(* Logix 5000 project; controller WWTP_SOLIDS_CLX vendor 1 type 14 code 54 rev 17.2; software revision 17.00; part 6 of 16 *)
(* tags used below, declared in another part *)
   Cfg_ClearPulseT : DINT;   // Time to pulse Out_Clear to clear external totalizer (sec)
   PCmd_ClearTot : BOOL;   // Program Command to Clear Totalizer Qty
   PCmd_StartTot : BOOL;   // Program Command to Start Totalizer
   PCmd_StopTot : BOOL;   // Program Command to Stop Totalizer
   PCmd_ZeroFaultInhibit : BOOL;   // Program Command to Inhibit Zero Fault Alarm
   PCmd_ZeroFaultUninhibit : BOOL;   // Program Command to Uninhibit Zero Fault Alarm
   OCmd_ClearTot : BOOL;   // Operator Command to Clear Totalizer Qty
   OCmd_StartTot : BOOL;   // Operator Command to Start Totalizer
   OCmd_StopTot : BOOL;   // Operator Command to Stop Totalizer
   Rdy_ClearTot : BOOL;   // 1=Ready for OCmd_ClearTot (enables button)
   Rdy_StartTot : BOOL;   // 1=Ready for OCmd_StartTot (enables button)
   Rdy_StopTot : BOOL;   // 1=Ready for OCmd_StopTot (enables button)
   Wrk_ValidONS : BOOL;   // Rate PV goes from Infinite or Not a Number to VALID
(* P_DoseFM, continued *)

ROUTINE Prescan   (* ladder *)
// Clear Ownership, clear "lurking" Commands, all Readies
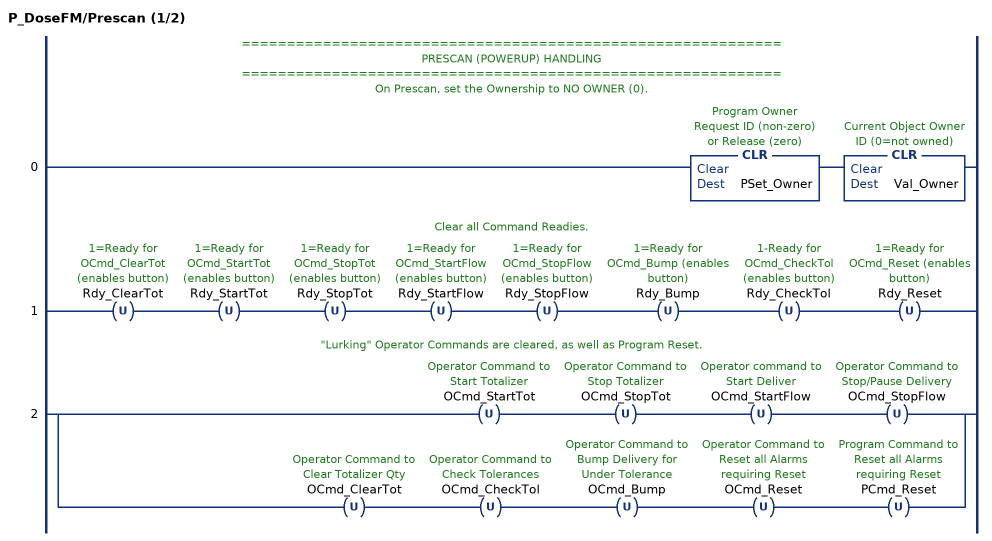
   // ============================================================
   // PRESCAN (POWERUP) HANDLING
   // ============================================================
   // On Prescan, set the Ownership to NO OWNER (0).
   0: CLR(PSet_Owner)CLR(Val_Owner);
   // Clear all Command Readies.
   1: OTU(Rdy_ClearTot)OTU(Rdy_StartTot)OTU(Rdy_StopTot)OTU(Rdy_StartFlow)OTU(Rdy_StopFlow)OTU(Rdy_Bump)OTU(Rdy_CheckTol)OTU(Rdy_Reset);
   // "Lurking" Operator Commands are cleared, as well as Program Reset.
   2: [OTU(OCmd_StartTot) OTU(OCmd_StopTot) OTU(OCmd_StartFlow) OTU(OCmd_StopFlow) ,OTU(OCmd_ClearTot) OTU(OCmd_CheckTol) OTU(OCmd_Bump) OTU(OCmd_Reset) OTU(PCmd_Reset) ];
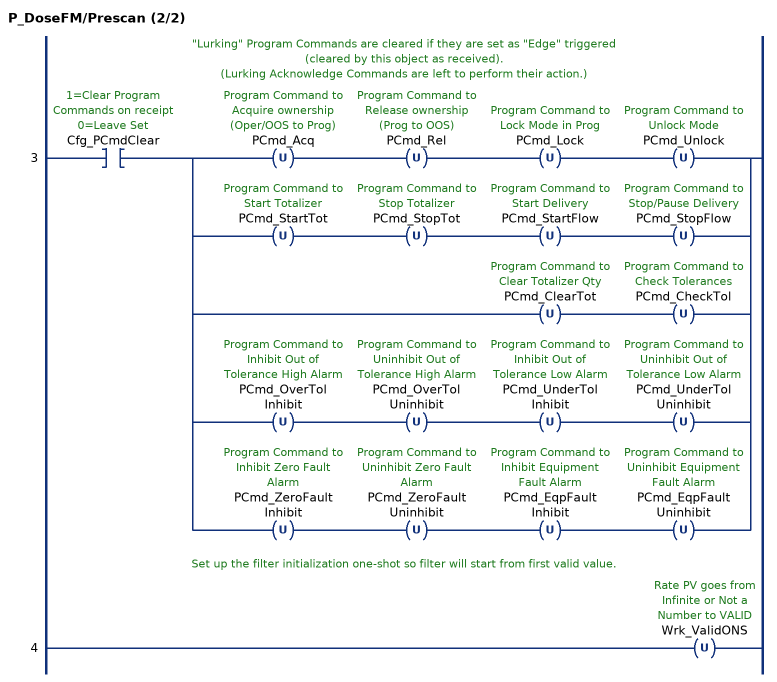
   // "Lurking" Program Commands are cleared if they are set as "Edge" triggered
   // (cleared by this object as received).
   // (Lurking Acknowledge Commands are left to perform their action.)
   3: XIC(Cfg_PCmdClear)[OTU(PCmd_Acq) OTU(PCmd_Rel) OTU(PCmd_Lock) OTU(PCmd_Unlock) ,OTU(PCmd_StartTot) OTU(PCmd_StopTot) OTU(PCmd_StartFlow) OTU(PCmd_StopFlow) ,OTU(PCmd_ClearTot) OTU(PCmd_CheckTol) ,OTU(PCmd_OverTolInhibit) OTU(PCmd_OverTolUninhibit) OTU(PCmd_UnderTolInhibit) OTU(PCmd_UnderTolUninhibit) ,OTU(PCmd_ZeroFaultInhibit) OTU(PCmd_ZeroFaultUninhibit) OTU(PCmd_EqpFaultInhibit) OTU(PCmd_EqpFaultUninhibit) ];
   // Set up the filter initialization one-shot so filter will start from first valid value.
   4: OTU(Wrk_ValidONS);
END_ROUTINE
END_ADD_ON_INSTRUCTION

ADD_ON_INSTRUCTION P_DoseWS   (* revision 0.8, ExecutePrescan, ExecuteEnableInFalse *)
// Dosing with Weigh Scale
// Revision note:
// Fixed handling of Infinite / Not a Number weight PV
// Help:
// This Instruction monitors a weigh scale and provides:
// *  Monitoring of weight rate of change to determine a flow Rate
// *  Command to Tare the scale (set the delivered Quantity to zero)
// *  Commands to Start and Stop Flow for a dosing
// *  Optional switching to a slow delivery (dribble) when approaching setpoint
// *  Stopping flow just before reaching setpoint using a Preact value
// *  Optional automatic adjustment of the preact value to fine tune the stop point
// *  Commands to check if the delivered quantity is within user-specified tolerances and alarm if not
// *  Program and Operator Settings for Setpoint, Preact, Dribble Quantity, High and Low Tolerances
// *  Equipment Failure Alarm on sensor or controlled equipment failure (stops flow)
// *  Tare failure alarm if scale does not stay at steady weight when tared
// *  Configurable Low Rate Cutoff to report zero Rate when scale rate of change is small
// *  Mode selection (Operator, Program or Maintenance)
// *  Simulation using simulated starting weight (Tare point), Running Rate and Dribble Rate
VAR_INPUT
   Inp_WeightPV : REAL; {visible}   // Weight from Weigh Scale (unscaled)
   Inp_PVBad : BOOL;   // 1=Scale PV or I/O Quality Bad, 0=OK
   Inp_PVUncertain : BOOL;   // 1=Scale PV Quality Uncertain, 0=OK
   Inp_CtrldEqpFault : BOOL; {visible}   // Controlled Equipment device or I/O status 0=OK, 1=fail
   Inp_Sim : BOOL;   // 1=Simulate working weigh scale; 0=use actual weight input
   Inp_Reset : BOOL; {visible}   // 1=Reset all fault conditions and latched Alarms
   Cfg_LossInWeight : BOOL;   // 1=Running reduces weight (Xfer Out), 0=iRunning ncreases weight (Xfer In)
   Cfg_HasDribble : BOOL;   // 1=Slow to Dribble before complete, 0=use complete only
   Cfg_AutoAdjPreact : BOOL;   // 1=enable automatic adjustment of preact after each delivery
   Cfg_SetTrack : BOOL := 1;   // 1=PSets track OSets in Oper, OSets track PSets in Prog, 0=no tracking
   Cfg_PCmdClear : BOOL := 1;   // 1=Clear Program Commands on receipt 0=Leave Set
   Cfg_HasOverTolAlm : BOOL;   // 1=Over Tolerance Alarm exists and will be checked
   Cfg_HasUnderTolAlm : BOOL;   // 1=Under Tolerance Alarm exists and will be checked
   Cfg_HasTareFaultAlm : BOOL;   // 1=Tare Fault Alarm exists and will be checked
   Cfg_HasEqpFaultAlm : BOOL;   // 1=Equipment Fault Alarm exists and will be checked
   Cfg_OverTolResetReqd : BOOL;   // 1=Reset requied to clear Out of Tolerance High Alarm
   Cfg_UnderTolResetReqd : BOOL;   // 1=Reset required to clear Out of Tolerance Low Alarm
   Cfg_TareFaultResetReqd : BOOL;   // 1=Reset required to clear Tare Fault Alarm
   Cfg_EqpFaultResetReqd : BOOL;   // 1=Reset required to clear Equipment Fault Alarm
   Cfg_OverTolAckReqd : BOOL := 1;   // 1=Acknowledge required for Out of Tolerance High Alarm
   Cfg_UnderTolAckReqd : BOOL := 1;   // 1=Acknowledge required for Out of Tolerance Low Alarm
   Cfg_TareFaultAckReqd : BOOL := 1;   // 1=Acknowledge required for Tare Fault Alarm
   Cfg_EqpFaultAckReqd : BOOL := 1;   // 1=Acknowledge required for Equipment Fault Alarm
   Cfg_OverTolSeverity : SINT := 3;   // Over Tolerance Alarm Severity 1=info, 2=warn, 3=excep, 4=fault
   Cfg_UnderTolSeverity : SINT := 2;   // Under Tolerance Alarm Severity 1=info, 2=warn, 3=excep, 4=fault
   Cfg_TareFaultSeverity : SINT := 4;   // Tare Fault Alarm Severity 1=info, 2=warn, 3=excep, 4=fault
   Cfg_EqpFaultSeverity : SINT := 4;   // Equipment Fault Alarm Severity 1=info, 2=warn, 3=excep, 4=fault
   Cfg_InpRawMin : REAL;   // Minimum unscaled weight input
   Cfg_InpRawMax : REAL := 10000.0;   // Maximum unscaled weight input
   Cfg_PVEUMin : REAL;   // Minimum scaled weight PV input (EU)
   Cfg_PVEUMax : REAL := 10000.0;   // Maximum scaled weight PV input (EU)
   Cfg_MaxQty : REAL := 1.e+38;   // Maximum allowed quantity to deliver (setpoint) (EU)
   Cfg_RateTime : REAL := 1.0;   // Time factor for rate (60 for /min, 3600 for /hr) (Sec)
   Cfg_RateFiltTC : REAL := 0.1;   // Filter Time Constant (sec) for calculated Rate
   Cfg_TareFaultLim : REAL := 1.0;   // Amount (EU) scale can drift after Tare before starting flow without Faulting
   Cfg_BumpT : REAL := 3.0;   // Bump (manual top-off) Time (Sec)
   Cfg_AutoAdjPct : REAL := 10.0;   // Percentage of delivery error to auto-adjust preact (%)
   Cfg_SimStartWt : REAL;   // Weight to start from (tare to) in simulation (EU)
   Cfg_SimRate : REAL := 1.0;   // Rate at which to deliver when running in Simulation (EU/rate time)
   Cfg_SimDribbleRate : REAL := 0.1;   // Rate at which to dribble when running in Simulation (EU/rate time)
   PSet_SP : REAL;   // Program Setting of total quantity to deliver (EU)
   PSet_DribbleQty : REAL;   // Program Setting of quantity to dribble (EU)
   PSet_Preact : REAL;   // Program Setting of amount before total to stop flow (EU)
   PSet_TolHi : REAL;   // Program Setting of High Tolerance Limit (OK amount > SP)
   PSet_TolLo : REAL;   // Program Setting of Low Tolerance Limit (OK amount < SP)
   PSet_Owner : DINT;   // Program Owner Request ID (non-zero) or Release (zero)
   OSet_SP : REAL;   // Operator Setting of total quantity to deliver (EU)
   OSet_DribbleQty : REAL;   // Operator Setting of quantity to dribble (EU)
   OSet_Preact : REAL;   // Operator Setting of amount before total to stop flow (EU)
   OSet_TolHi : REAL;   // Operator Setting of High Tolerance Limit (OK amount > SP)
   OSet_TolLo : REAL;   // Operator Setting of Low Tolerance Limit (OK amount < SP)
   PCmd_Tare : BOOL;   // Program Command to Tare (reset delivered qty to 0)
   PCmd_StartFlow : BOOL;   // Program Command to Start Delivery
   PCmd_StopFlow : BOOL;   // Program Command to Stop/Pause Delivery
   PCmd_CheckTol : BOOL;   // Program Command to Check Tolerances
   PCmd_Acq : BOOL;   // Program Command to Acquire ownership (Oper/OOS to Prog)
   PCmd_Rel : BOOL;   // Program Command to Release ownership (Prog to OOS)
   PCmd_Lock : BOOL;   // Program Command to Lock Mode in Prog
   PCmd_Unlock : BOOL;   // Program Command to Unlock Mode
   PCmd_Reset : BOOL;   // Program Command to Reset all Alarms requiring Reset
   PCmd_OverTolAck : BOOL;   // Program Command to Acknowledge Out of Tolerance High Alarm
   PCmd_OverTolInhibit : BOOL;   // Program Command to Inhibit Out of Tolerance High Alarm
   PCmd_OverTolUninhibit : BOOL;   // Program Command to Uninhibit Out of Tolerance High Alarm
   PCmd_UnderTolAck : BOOL;   // Program Command to Acknowledge Out of Tolerance Low Alarm
   PCmd_UnderTolInhibit : BOOL;   // Program Command to Inhibit Out of Tolerance Low Alarm
   PCmd_UnderTolUninhibit : BOOL;   // Program Command to Uninhibit Out of Tolerance Low Alarm
   PCmd_TareFaultAck : BOOL;   // Program Command to Acknowledge Tare Fault Alarm
   PCmd_TareFaultInhibit : BOOL;   // Program Command to Inhibit Tare Fault Alarm
   PCmd_TareFaultUninhibit : BOOL;   // Program Command to Uninhibit Tare Fault Alarm
   PCmd_EqpFaultAck : BOOL;   // Program Command to Acknowledge Equipment Fault Alarm
   PCmd_EqpFaultInhibit : BOOL;   // Program Command to Inhibit Equipment Fault Alarm
   PCmd_EqpFaultUninhibit : BOOL;   // Program Command to Uninhibit Equipment Fault Alarm
   OCmd_Tare : BOOL;   // Operator Command to Tare (reset delivered qty to 0)
   OCmd_StartFlow : BOOL;   // Operator command to Start Deliver
   OCmd_StopFlow : BOOL;   // Operator Command to Stop/Pause Delivery
   OCmd_CheckTol : BOOL;   // Operator Command to Check Tolerances
   OCmd_Bump : BOOL;   // Operator Command to Bump Delivery for Under Tolerance
   OCmd_Reset : BOOL;   // Operator Command to Reset all Alarms requiring Reset
END_VAR
VAR_OUTPUT
   Out_RunFlow : BOOL; {visible}   // 1=Deliver at Full (fast) Flow
   Out_DribbleFlow : BOOL; {visible}   // 1=Deliver at Dribble (slow) Flow
   Out_StopFlow : BOOL; {visible}   // 1=Stop Delivery Equipment
   Val_PV : REAL; {visible}   // Weight on Scale (EU)
   Val_Tare : REAL; {visible}   // Weight on Scale when Tare Command received (EU)
   Val_Qty : REAL; {visible}   // Quantity actually delivered (totalizer output) (EU)
   Val_Rate : REAL; {visible}   // Current Delivery Rate (EU/time) (see Cfg_RateTime)
   Val_SP : REAL; {visible}   // Amount to be delivered (Setpoint) (EU)
   Val_Remain : REAL; {visible}   // Amount yet to deliver to reach Setpoint (EU)
   Val_PctComplete : REAL; {visible}   // Percent Complete (for Progress Bar on HMI) 0.0 to 100.0%
   Val_DribbleQty : REAL; {visible}   // Amount to be delivered at slow rate (EU)
   Val_Preact : REAL; {visible}   // Amount before SP at which flow will be stopped (EU)
   Val_TolHi : REAL; {visible}   // Allowed Amount > SP (EU)
   Val_TolLo : REAL; {visible}   // Allowed Amount < SP (EU)
   Val_PVEUMin : REAL;   // Minimum of scaled range = MIN (Cfg_PVEUMin, Cfg_PVEUMax)
   Val_PVEUMax : REAL := 10000.0;   // Maximum of scaled range = MAX (Cfg_PVEUMin, Cfg_PVEUMax)
   Val_Owner : DINT;   // Current Object Owner ID (0=not owned)
   Val_Notify : SINT;   // Current Alarm Level and Acknowledgement (enumeration)
   Sts_Tared : BOOL; {visible}   // Scale Tare completed, Qty = 0.0
   Sts_FlowRunning : BOOL; {visible}   // 1=Flow is Running (Out_Run is ON)
   Sts_FlowDribble : BOOL; {visible}   // 1=Flow is slowed to Dribble (Out_Dribble is ON)
   Sts_FlowStopped : BOOL; {visible}   // 1=Flow is Stopped (Out_Stop is ON)
   Sts_Bumping : BOOL;   // 1=Bump flow (timed) is active
   Sts_Complete : BOOL; {visible}   // 1=Total Delivered > (SP - Preact)
   Sts_InTol : BOOL;   // 1=Total Delivered is Within Tolerances
   Sts_Available : BOOL;   // 1=Dosing available for control by automation (Prog)
   Sts_PVBad : BOOL;   // 1=Weight PV and Rate PV Quality Bad (I/O fail), 0=OK
   Sts_PVUncertain : BOOL;   // 1=Weight PV and Rate PV Quality is Uncertian, 0=OK
   Sts_Err : BOOL; {visible}   // 1=Error: Bad Configuration, see detail Err bits for reason
   Err_Raw : BOOL;   // 1=Error: Cfg_InpRawMax or Cfg_InpRawMin invalid
   Err_EU : BOOL;   // 1=Error: Cfg_PVEUMax or Cfg_PVEUMin invalid
   Err_Rate : BOOL;   // 1=Error: Cfg_RateFiltTC or Cfg_RateTime invalid
   Err_Limit : BOOL;   // 1=Error: Cfg_MaxQty invalid
   Err_Sim : BOOL;   // 1=Error: Cfg_SimDribbleRate or Cfg_SimRate invalid
   Err_Timer : BOOL;   // 1=Error: Cfg_BumpT (use 0.0 to 2147483.647)
   Err_Alarm : BOOL;   // 1=Error: Alarm Min Duration or Severity Cfg Invalid
   Sts_Maint : BOOL; {visible}   // 1=Mode is Maintenance (supersedes Prog, Oper)
   Sts_Prog : BOOL; {visible}   // 1=Mode is Program (auto)
   Sts_Oper : BOOL := 1; {visible}   // 1=Mode is Operator (manual)
   Sts_ProgOperLock : BOOL;   // 1=Program or Operator has requested Mode Lock
   Sts_OverTol : BOOL;   // 1=Delivery Out of Tolerance High
   Alm_OverTol : BOOL;   // 1=Delivery Out of Tolerance High Alarm
   Ack_OverTol : BOOL;   // 1=Out of Tolerance High Alarm has been acknowledged
   Sts_OverTolDisabled : BOOL;   // 1=Out of Tolerance High Alarm has been disabled (will not be sent)
   Sts_OverTolInhibited : BOOL;   // 1=Out of Tolerance High Alarm has been inhibited by logic
   Sts_OverTolSuppressed : BOOL;   // 1=Out of Tolerance High Alarm has been suppressed (logged only)
   Sts_UnderTol : BOOL;   // 1=Delivery Out of Tolerance Low
   Alm_UnderTol : BOOL;   // 1=Delivery Out of Tolerance Low Alarm
   Ack_UnderTol : BOOL;   // 1=Out of Tolerance Low Alarm has been acknowledged
   Sts_UnderTolDisabled : BOOL;   // 1=Out of Tolerance Low Alarm has been disabled (will not be sent)
   Sts_UnderTolInhibited : BOOL;   // 1=Out of Tolerance Low Alarm has been inhibited by logic
   Sts_UnderTolSuppressed : BOOL;   // 1=Out of Tolerance Low Alarm has been suppressed (logged only)
   Sts_TareFault : BOOL;   // 1=Scale reading moved unexpectedly since Tare
   Alm_TareFault : BOOL;   // 1=Warning: scale reading moved since Tare
   Ack_TareFault : BOOL;   // 1=Tare Fault Alarm has been acknowledged
   Sts_TareFaultDisabled : BOOL;   // 1=Tare Fault Alarm is Disabled (not saved or sent)
   Sts_TareFaultInhibited : BOOL;   // 1=Tare Fault Alarm has been inhibited by logic
   Sts_TareFaultSuppressed : BOOL;   // 1=Tare Fault Alarm has been suppressed (logged only)
   Sts_EqpFault : BOOL;   // 1=Equipment Fault Detected
   Alm_EqpFault : BOOL;   // 1=Equipment Fault Alarm
   Ack_EqpFault : BOOL;   // 1=Equipment Fault Alarm has been acknowledged
   Sts_EqpFaultDisabled : BOOL;   // 1=Equipment Fault Alarm is Disabled (not saved or sent)
   Sts_EqpFaultInhibited : BOOL;   // 1=Equipment Fault Alarm has been inhibited by logic
   Sts_EqpFaultSuppressed : BOOL;   // 1=Equipment Fault Alarm has been suppressed (logged only)
   Rdy_Tare : BOOL;   // 1=Ready for OCmd_Tare (enables button)
   Rdy_StartFlow : BOOL;   // 1=Ready for OCmd_StartFlow (enables button)
   Rdy_StopFlow : BOOL;   // 1=Ready for OCmd_StopFlow (enables button)
   Rdy_CheckTol : BOOL;   // 1-Ready for OCmd_CheckTol (enables button)
   Rdy_Bump : BOOL;   // 1=Ready for OCmd_Bump (enables button)
   Rdy_Reset : BOOL;   // 1=Ready for OCmd_Reset (enables button)
END_VAR
VAR
   Cfg_RateEU : STRING_8 := 'kg/sec';   // Engineering Units for Rate (flow) for display on HMI
   Cfg_Tag : STRING_20 := 'P_DoseWS';   // Tagname for display on HMI
   Cfg_Label : STRING_20 := 'Weigh Scale Dosing';   // Label for graphic symbol displayed on HMI
   Cfg_QtyEU : STRING_8 := 'kg';   // Engineering Units for Quantity for display on HMI
   Cfg_Desc : STRING_40 := 'Dosing with Weigh Scale';   // Description for display on HMI
   Wrk_Notify : DINT;   // Buffer for building Val_Notify
   Mode : P_Mode := (Cfg_PCmdClear := 1, Cfg_OvrdOverLock := 1, Sts_Oper := 1, Rdy_Rel := 1, Rdy_AcqLock := 1);   // Analog Input Mode Selection
   Wrk_Tare : BOOL;   // Request to Tare Scale received
   TareFault : P_Alarm := (Inp := 1, Cfg_AckReqd := 1, Cfg_Severity := 3, Ack := 1, Rdy_Disable := 1);   // Scale not holding at point at which Tared Alarm
   UnderTol : P_Alarm := (Inp := 1, Cfg_AckReqd := 1, Cfg_Severity := 3, Ack := 1, Rdy_Disable := 1);   // Final Quantity Below Low Tolerance Alarm
   OverTol : P_Alarm := (Inp := 1, Cfg_AckReqd := 1, Cfg_Severity := 3, Ack := 1, Rdy_Disable := 1);   // Final Quantity Above High Tolerance Alarm
   EqpFault : P_Alarm := (Inp := 1, Cfg_AckReqd := 1, Cfg_Severity := 3, Ack := 1, Rdy_Disable := 1);   // Equipment (Sensor, Controlled Equip.) Fault Alarm
   Wrk_RunFlow : BOOL;   // 1=Flow (full)( should be running
   Wrk_BumpFlow : BOOL;   // Operator requested bump flow to make up Under Tolerance
   Wrk_BumpT : TIMER := (PRE := 3000);   // Bump Timer for shot of flow to make up Under Tolerance
   Wrk_ScanTime : REAL;   // Time since previous scan (sec)
   Wrk_PrevPV : REAL;   // Previous scan's Val_PV value
   Wrk_Rate : REAL;   // Instantaneous Rate based on change in Inp_Qty
   Wrk_AmtToAdd : REAL;   // Amount to add to Quantity this scan based on Rate
   Wrk_PctComplete : REAL;   // Percent Complete calculation intermediate
   Wrk_PV : REAL;   // Working value of Scale Weight (actual or simulated)
   Wrk_TareWt : REAL;   // Weight on scale when Tare Command received
   Wrk_FiltRate : REAL;   // Working register for calculating filtered delivery rate
   Wrk_BumpNoAdj : BOOL;   // Do NOT auto-adjust Preact if flow was Bumped since Tare
   Wrk_ScanT : TIMER := (PRE := 2147483647);   // Scan Timer (milliseconds, always runs)
   Wrk_Alpha : REAL;   // Filter multiplier = (1 / (1+TC/dT) )
   Wrk_InpDINT : DINT;   // Inp_WeightPV check for Infinite or Not A Number
   Wrk_InpInfNaN : BOOL;   // Input Weight is Infinite or NaN
   Wrk_ValidONS1 : BOOL;   // Weight PV goes from Infinite or Not a Number to VALID
   Wrk_ValidONS2 : BOOL;   // Rate goes from Infinite or Not a Number to VALID
END_VAR

ROUTINE EnableInFalse   (* ladder *)
// Clear any "lurking" Commands and all Readies, set NO MODE
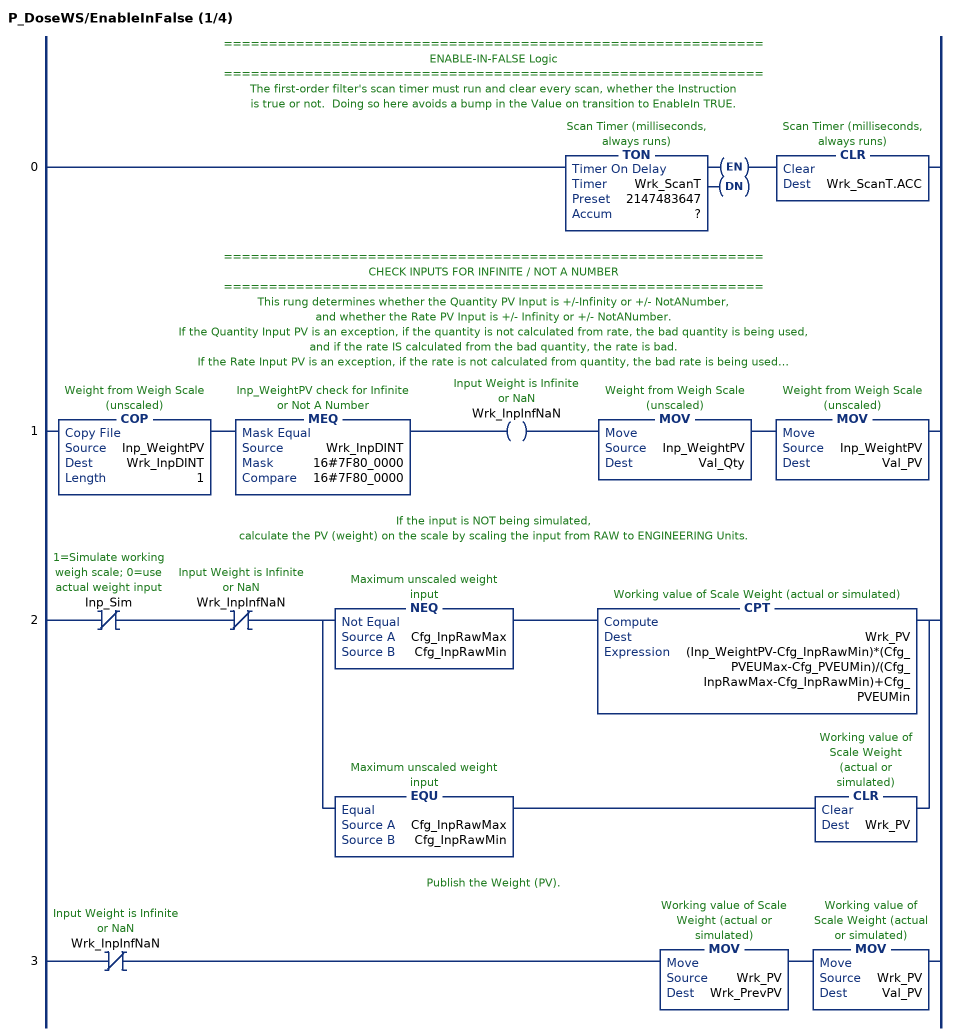
   // ============================================================
   // ENABLE-IN-FALSE Logic
   // ============================================================
   // The first-order filter's scan timer must run and clear every scan, whether the Instruction
   // is true or not.  Doing so here avoids a bump in the Value on transition to EnableIn TRUE.
   0: TON(Wrk_ScanT,?,?)CLR(Wrk_ScanT.ACC);
   // ============================================================
   // CHECK INPUTS FOR INFINITE / NOT A NUMBER
   // ============================================================
   // This rung determines whether the Quantity PV Input is +/-Infinity or +/- NotANumber,
   // and whether the Rate PV Input is +/- Infinity or +/- NotANumber.
   // If the Quantity Input PV is an exception, if the quantity is not calculated from rate, the bad quantity is being used,
   // and if the rate IS calculated from the bad quantity, the rate is bad.
   // If the Rate Input PV is an exception, if the rate is not calculated from quantity, the bad rate is being used,
   // and if the quantity IS calculated from the bad rate, the quantity is bad.
   1: COP(Inp_WeightPV,Wrk_InpDINT,1)MEQ(Wrk_InpDINT,16#7F80_0000,16#7F80_0000)OTE(Wrk_InpInfNaN)MOV(Inp_WeightPV,Val_Qty)MOV(Inp_WeightPV,Val_PV);
   // If the input is NOT being simulated,
   // calculate the PV (weight) on the scale by scaling the input from RAW to ENGINEERING Units.
   2: XIO(Inp_Sim)XIO(Wrk_InpInfNaN)[NEQ(Cfg_InpRawMax,Cfg_InpRawMin) CPT(Wrk_PV,(Inp_WeightPV-Cfg_InpRawMin)*(Cfg_PVEUMax-Cfg_PVEUMin)/(Cfg_InpRawMax-Cfg_InpRawMin)+Cfg_PVEUMin) ,EQU(Cfg_InpRawMax,Cfg_InpRawMin) CLR(Wrk_PV) ];
   // Publish the Weight (PV).
   3: XIO(Wrk_InpInfNaN)MOV(Wrk_PV,Wrk_PrevPV)MOV(Wrk_PV,Val_PV);
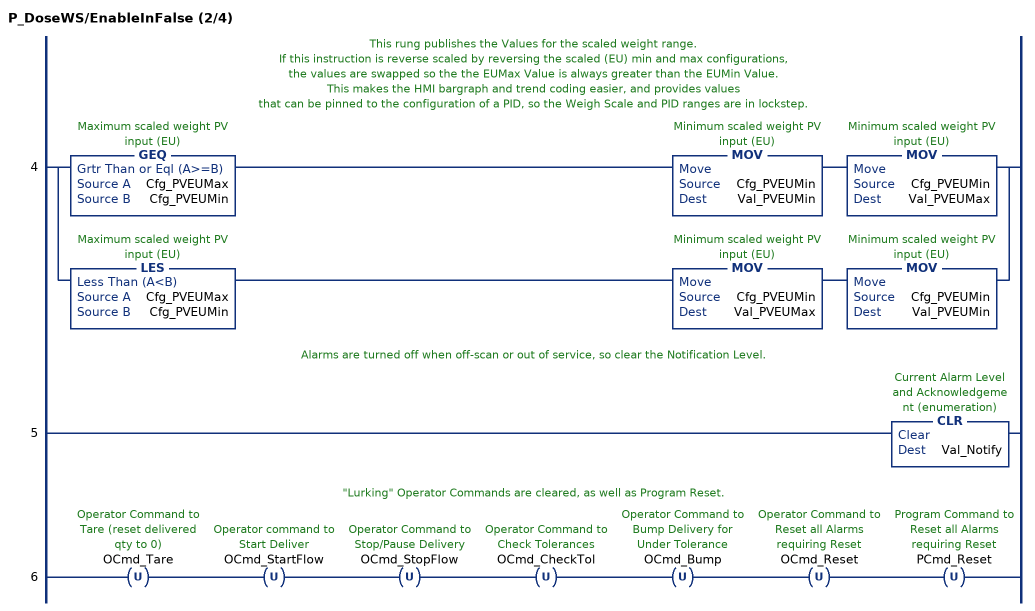
   // This rung publishes the Values for the scaled weight range.
   // If this instruction is reverse scaled by reversing the scaled (EU) min and max configurations,
   // the values are swapped so the the EUMax Value is always greater than the EUMin Value.
   // This makes the HMI bargraph and trend coding easier, and provides values
   // that can be pinned to the configuration of a PID, so the Weigh Scale and PID ranges are in lockstep.
   4: [GEQ(Cfg_PVEUMax,Cfg_PVEUMin) MOV(Cfg_PVEUMin,Val_PVEUMin) MOV(Cfg_PVEUMin,Val_PVEUMax) ,LES(Cfg_PVEUMax,Cfg_PVEUMin) MOV(Cfg_PVEUMin,Val_PVEUMax) MOV(Cfg_PVEUMin,Val_PVEUMin) ];
   // Alarms are turned off when off-scan or out of service, so clear the Notification Level.
   5: CLR(Val_Notify);
   // "Lurking" Operator Commands are cleared, as well as Program Reset.
   6: OTU(OCmd_Tare)OTU(OCmd_StartFlow)OTU(OCmd_StopFlow)OTU(OCmd_CheckTol)OTU(OCmd_Bump)OTU(OCmd_Reset)OTU(PCmd_Reset);
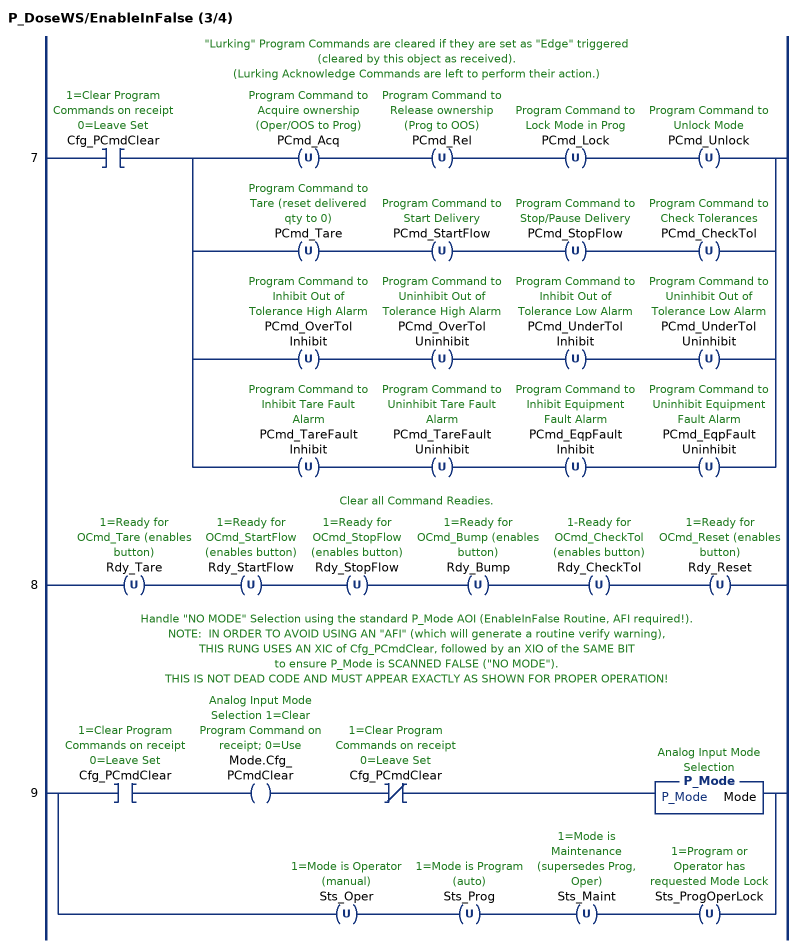
   // "Lurking" Program Commands are cleared if they are set as "Edge" triggered
   // (cleared by this object as received).
   // (Lurking Acknowledge Commands are left to perform their action.)
   7: XIC(Cfg_PCmdClear)[OTU(PCmd_Acq) OTU(PCmd_Rel) OTU(PCmd_Lock) OTU(PCmd_Unlock) ,OTU(PCmd_Tare) OTU(PCmd_StartFlow) OTU(PCmd_StopFlow) OTU(PCmd_CheckTol) ,OTU(PCmd_OverTolInhibit) OTU(PCmd_OverTolUninhibit) OTU(PCmd_UnderTolInhibit) OTU(PCmd_UnderTolUninhibit) ,OTU(PCmd_TareFaultInhibit) OTU(PCmd_TareFaultUninhibit) OTU(PCmd_EqpFaultInhibit) OTU(PCmd_EqpFaultUninhibit) ];
   // Clear all Command Readies.
   8: OTU(Rdy_Tare)OTU(Rdy_StartFlow)OTU(Rdy_StopFlow)OTU(Rdy_Bump)OTU(Rdy_CheckTol)OTU(Rdy_Reset);
   // Handle "NO MODE" Selection using the standard P_Mode AOI (EnableInFalse Routine, AFI required!).
   // NOTE:  IN ORDER TO AVOID USING AN "AFI" (which will generate a routine verify warning),
   // THIS RUNG USES AN XIC of Cfg_PCmdClear, followed by an XIO of the SAME BIT
   // to ensure P_Mode is SCANNED FALSE ("NO MODE").
   // THIS IS NOT DEAD CODE AND MUST APPEAR EXACTLY AS SHOWN FOR PROPER OPERATION!
   9: [XIC(Cfg_PCmdClear) OTE(Mode.Cfg_PCmdClear) XIO(Cfg_PCmdClear) P_Mode(Mode) ,OTU(Sts_Oper) OTU(Sts_Prog) OTU(Sts_Maint) OTU(Sts_ProgOperLock) ];
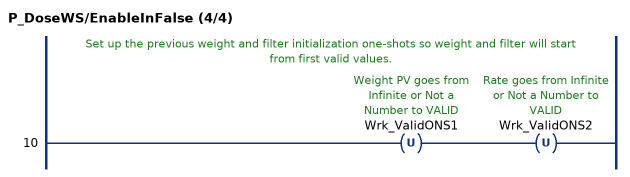
   // Set up the previous weight and filter initialization one-shots so weight and filter will start from first valid values.
   10: OTU(Wrk_ValidONS1)OTU(Wrk_ValidONS2);
END_ROUTINE

ROUTINE Logic   (* ladder *)
// Normal Scan: control / monitor Dosing with Weigh Scale
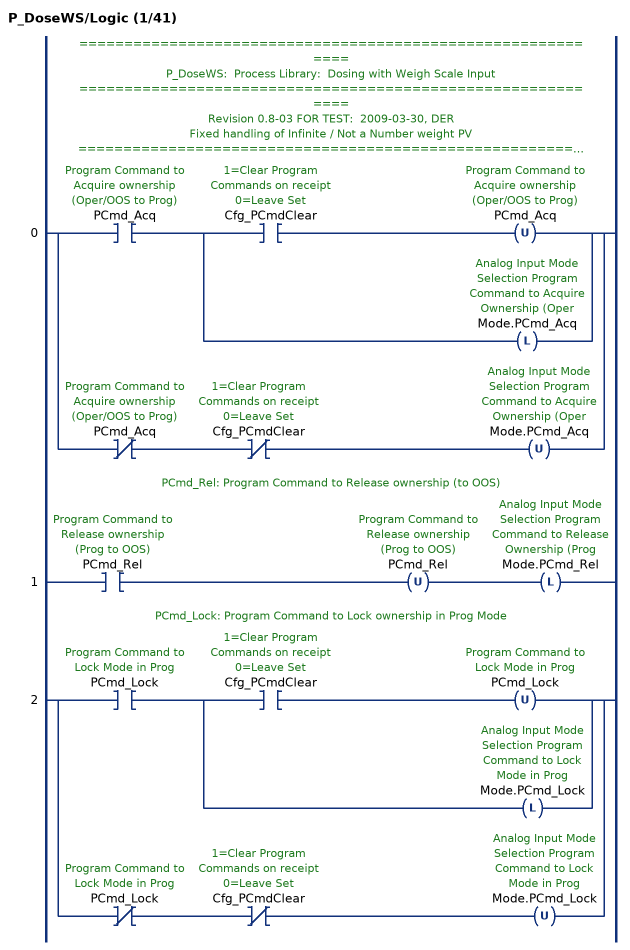
   // ============================================================
   // P_DoseWS:  Process Library:  Dosing with Weigh Scale Input
   // ============================================================
   // Revision 0.8-03 FOR TEST:  2009-03-30, DER
   // Fixed handling of Infinite / Not a Number weight PV
   // ============================================================
   // This Instruction monitors a weigh scale and provides:
   // *  Monitor weight rate of change to determine a flow Rate
   // *  Command to Tare the scale (set the delivered Quantity to zero)
   // *  Commands to Start and Stop Flow for a dosing
   // *  Optional switching to a slow delivery (dribble) when approaching setpoint
   // *  Stopping flow just before reaching setpoint using a Preact value
   // *  Optional automatic adjustment of the preact value to fine tune the stop point
   // *  Commands to check if the delivered quantity is within user-specified tolerances and alarm if not
   // *  Program and Operator Settings for Setpoint, Preact, Dribble Quantity, High and Low Tolerances
   // *  Equipment Failure Alarm on sensor or controlled equipment failure (stops flow)
   // *  Tare failure alarm if scale does not stay at steady weight when tared
   // *  Configurable Low Rate Cutoff to report zero Rate when scale rate of change is small
   // *  Mode selection (Operator, Program or Maintenance)
   // *  Simulation using a provided simulated Tare point, Running Rate and Dribble Rate
   // ============================================================
   // POWERUP / INVALID STATE HANDLING
   // ============================================================
   // See the Prescan routine for powerup handling.
   // Mode states are retained through a power cycle.
   // ============================================================
   // MODE PROCESSING
   // ============================================================
   // These rungs handle received Mode Inputs and Commands:
   // NOTE:  Operator Commands for Mode, Alarm are sent directly to the contained P_Mode and P_Alarm AOIs.
   // PCmd_Acq: Program Command to Acquire ownership
   0: [XIC(PCmd_Acq) [XIC(Cfg_PCmdClear) OTU(PCmd_Acq) ,OTL(Mode.PCmd_Acq) ] ,XIO(PCmd_Acq) XIO(Cfg_PCmdClear) OTU(Mode.PCmd_Acq) ];
   // PCmd_Rel: Program Command to Release ownership (to OOS)
   1: XIC(PCmd_Rel)OTU(PCmd_Rel)OTL(Mode.PCmd_Rel);
   // PCmd_Lock: Program Command to Lock ownership in Prog Mode
   2: [XIC(PCmd_Lock) [XIC(Cfg_PCmdClear) OTU(PCmd_Lock) ,OTL(Mode.PCmd_Lock) ] ,XIO(PCmd_Lock) XIO(Cfg_PCmdClear) OTU(Mode.PCmd_Lock) ];
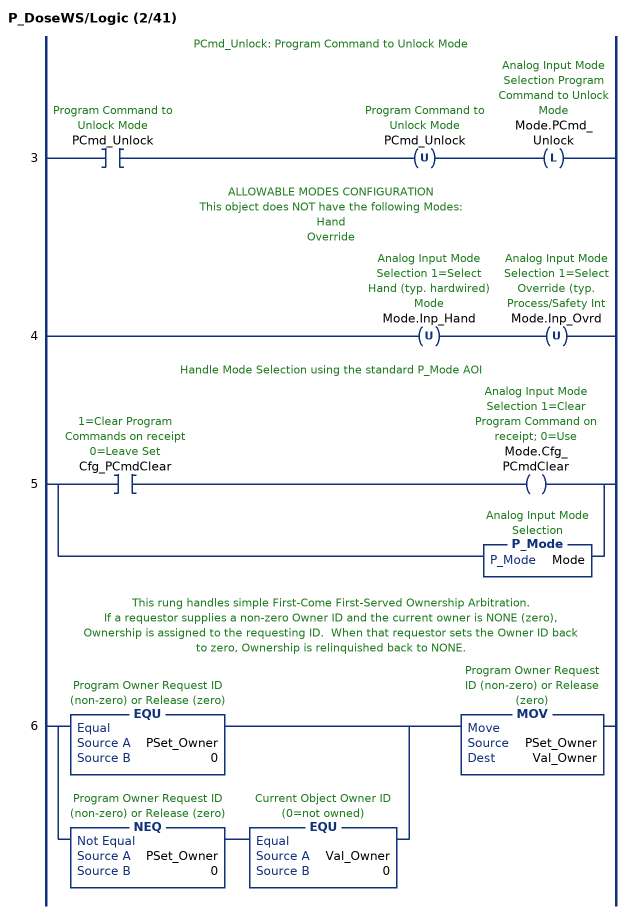
   // PCmd_Unlock: Program Command to Unlock Mode
   3: XIC(PCmd_Unlock)OTU(PCmd_Unlock)OTL(Mode.PCmd_Unlock);
   // ALLOWABLE MODES CONFIGURATION
   // This object does NOT have the following Modes:
   // Hand
   // Override
   4: OTU(Mode.Inp_Hand)OTU(Mode.Inp_Ovrd);
   // Handle Mode Selection using the standard P_Mode AOI
   5: [XIC(Cfg_PCmdClear) OTE(Mode.Cfg_PCmdClear) ,P_Mode(Mode) ];
   // This rung handles simple First-Come First-Served Ownership Arbitration.
   // If a requestor supplies a non-zero Owner ID and the current owner is NONE (zero),
   // Ownership is assigned to the requesting ID.  When that requestor sets the Owner ID back
   // to zero, Ownership is relinquished back to NONE.
   6: [EQU(PSet_Owner,0) ,NEQ(PSet_Owner,0) EQU(Val_Owner,0) ]MOV(PSet_Owner,Val_Owner);
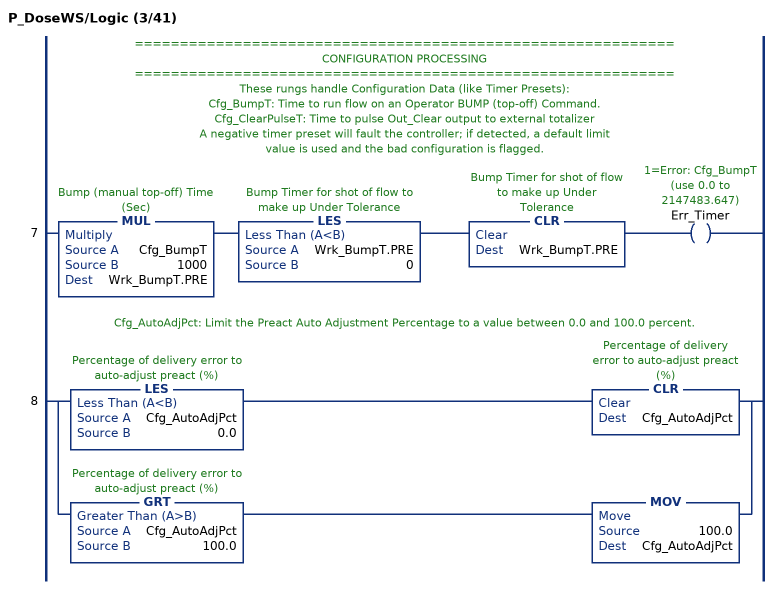
   // ============================================================
   // CONFIGURATION PROCESSING
   // ============================================================
   // These rungs handle Configuration Data (like Timer Presets):
   // Cfg_BumpT: Time to run flow on an Operator BUMP (top-off) Command.
   // Cfg_ClearPulseT: Time to pulse Out_Clear output to external totalizer
   // A negative timer preset will fault the controller; if detected, a default limit
   // value is used and the bad configuration is flagged.
   7: MUL(Cfg_BumpT,1000,Wrk_BumpT.PRE)LES(Wrk_BumpT.PRE,0)CLR(Wrk_BumpT.PRE)OTE(Err_Timer);
   // Cfg_AutoAdjPct: Limit the Preact Auto Adjustment Percentage to a value between 0.0 and 100.0 percent.
   8: [LES(Cfg_AutoAdjPct,0.0) CLR(Cfg_AutoAdjPct) ,GRT(Cfg_AutoAdjPct,100.0) MOV(100.0,Cfg_AutoAdjPct) ];
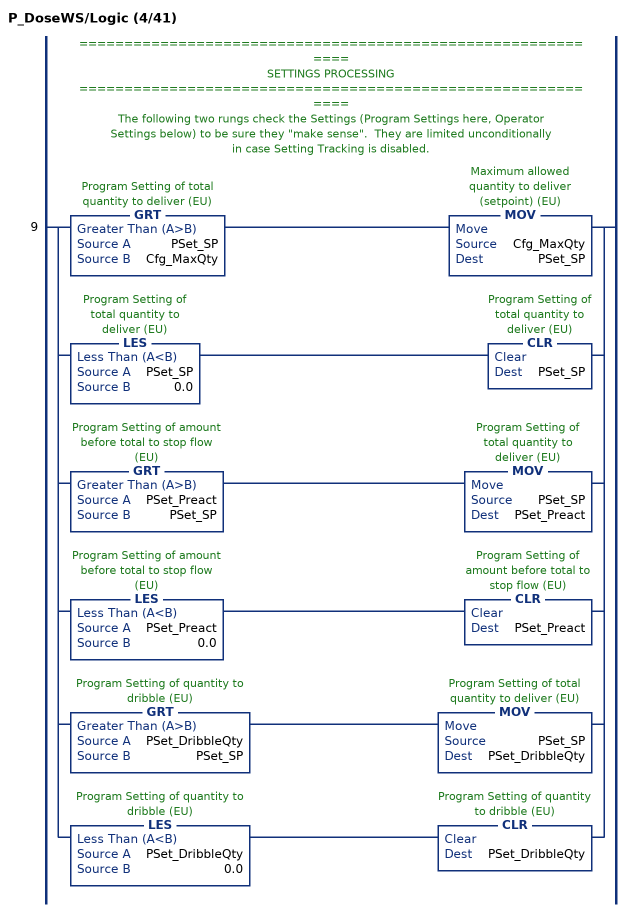
   // ============================================================
   // SETTINGS PROCESSING
   // ============================================================
   // The following two rungs check the Settings (Program Settings here, Operator
   // Settings below) to be sure they "make sense".  They are limited unconditionally
   // in case Setting Tracking is disabled.
   9: [GRT(PSet_SP,Cfg_MaxQty) MOV(Cfg_MaxQty,PSet_SP) ,LES(PSet_SP,0.0) CLR(PSet_SP) ,GRT(PSet_Preact,PSet_SP) MOV(PSet_SP,PSet_Preact) ,LES(PSet_Preact,0.0) CLR(PSet_Preact) ,GRT(PSet_DribbleQty,PSet_SP) MOV(PSet_SP,PSet_DribbleQty) ,LES(PSet_DribbleQty,0.0) CLR(PSet_DribbleQty) ];
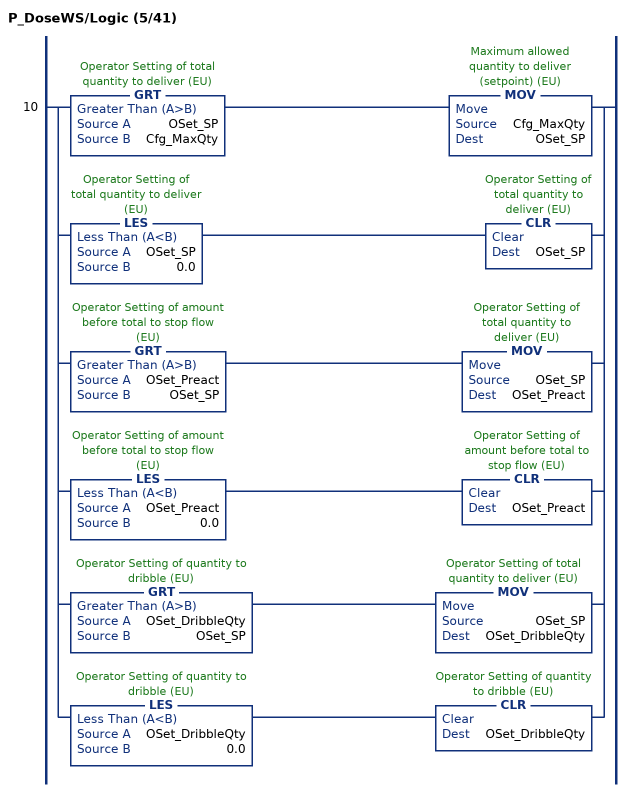
   10: [GRT(OSet_SP,Cfg_MaxQty) MOV(Cfg_MaxQty,OSet_SP) ,LES(OSet_SP,0.0) CLR(OSet_SP) ,GRT(OSet_Preact,OSet_SP) MOV(OSet_SP,OSet_Preact) ,LES(OSet_Preact,0.0) CLR(OSet_Preact) ,GRT(OSet_DribbleQty,OSet_SP) MOV(OSet_SP,OSet_DribbleQty) ,LES(OSet_DribbleQty,0.0) CLR(OSet_DribbleQty) ];
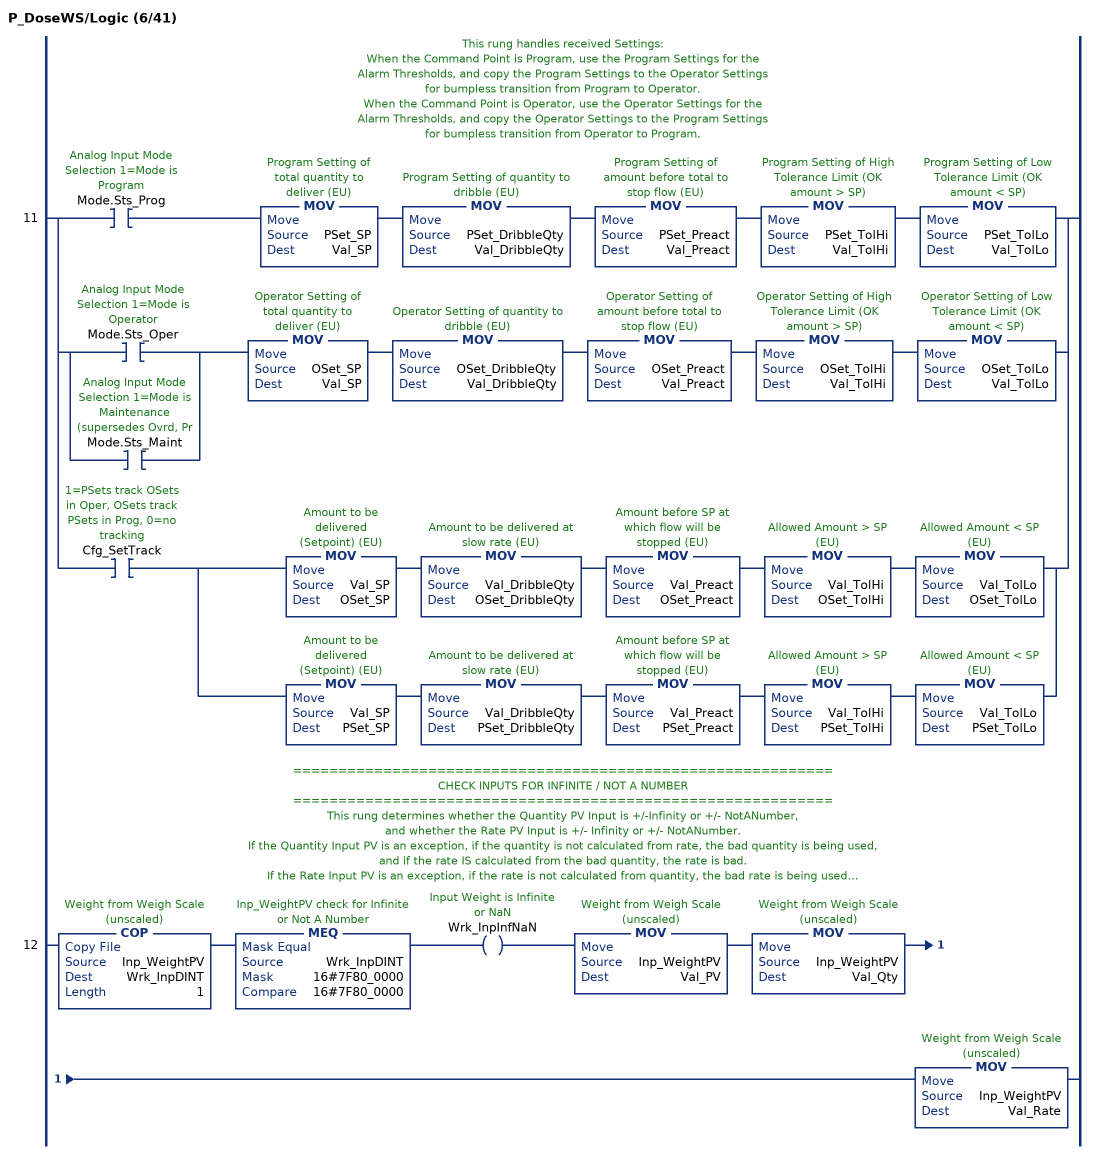
   // This rung handles received Settings:
   // When the Command Point is Program, use the Program Settings for the
   // Alarm Thresholds, and copy the Program Settings to the Operator Settings
   // for bumpless transition from Program to Operator.
   // When the Command Point is Operator, use the Operator Settings for the
   // Alarm Thresholds, and copy the Operator Settings to the Program Settings
   // for bumpless transition from Operator to Program.
   11: [XIC(Mode.Sts_Prog) MOV(PSet_SP,Val_SP) MOV(PSet_DribbleQty,Val_DribbleQty) MOV(PSet_Preact,Val_Preact) MOV(PSet_TolHi,Val_TolHi) MOV(PSet_TolLo,Val_TolLo) ,[XIC(Mode.Sts_Oper) ,XIC(Mode.Sts_Maint) ] MOV(OSet_SP,Val_SP) MOV(OSet_DribbleQty,Val_DribbleQty) MOV(OSet_Preact,Val_Preact) MOV(OSet_TolHi,Val_TolHi) MOV(OSet_TolLo,Val_TolLo) ,XIC(Cfg_SetTrack) [MOV(Val_SP,OSet_SP) MOV(Val_DribbleQty,OSet_DribbleQty) MOV(Val_Preact,OSet_Preact) MOV(Val_TolHi,OSet_TolHi) MOV(Val_TolLo,OSet_TolLo) ,MOV(Val_SP,PSet_SP) MOV(Val_DribbleQty,PSet_DribbleQty) MOV(Val_Preact,PSet_Preact) MOV(Val_TolHi,PSet_TolHi) MOV(Val_TolLo,PSet_TolLo) ] ];
   // ============================================================
   // CHECK INPUTS FOR INFINITE / NOT A NUMBER
   // ============================================================
   // This rung determines whether the Quantity PV Input is +/-Infinity or +/- NotANumber,
   // and whether the Rate PV Input is +/- Infinity or +/- NotANumber.
   // If the Quantity Input PV is an exception, if the quantity is not calculated from rate, the bad quantity is being used,
   // and if the rate IS calculated from the bad quantity, the rate is bad.
   // If the Rate Input PV is an exception, if the rate is not calculated from quantity, the bad rate is being used,
   // and if the quantity IS calculated from the bad rate, the quantity is bad.
   12: COP(Inp_WeightPV,Wrk_InpDINT,1)MEQ(Wrk_InpDINT,16#7F80_0000,16#7F80_0000)OTE(Wrk_InpInfNaN)MOV(Inp_WeightPV,Val_PV)MOV(Inp_WeightPV,Val_Qty)MOV(Inp_WeightPV,Val_Rate);
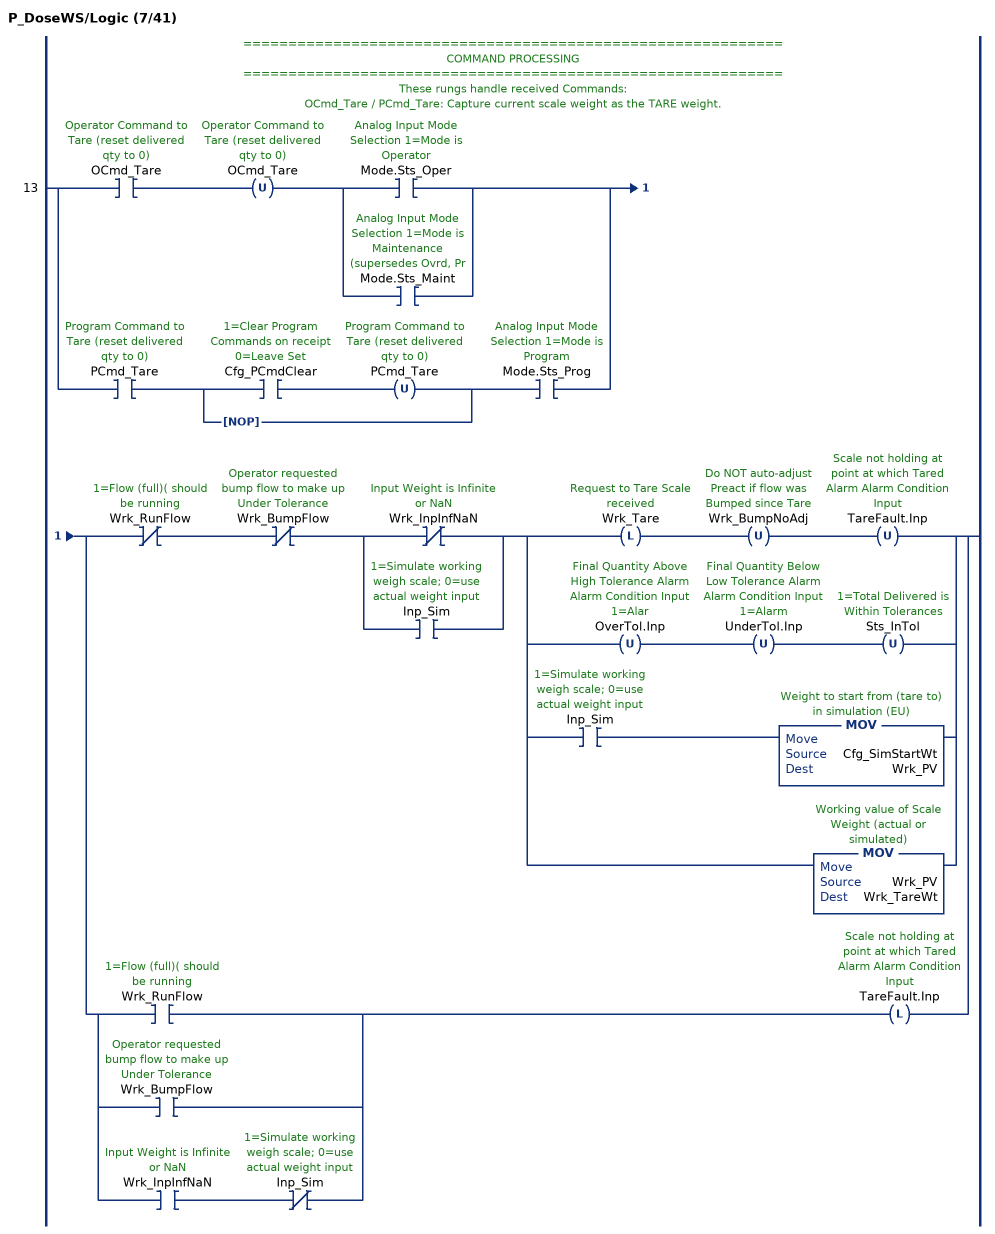
   // ============================================================
   // COMMAND PROCESSING
   // ============================================================
   // These rungs handle received Commands:
   // OCmd_Tare / PCmd_Tare: Capture current scale weight as the TARE weight.
   13: [XIC(OCmd_Tare) OTU(OCmd_Tare) [XIC(Mode.Sts_Oper) ,XIC(Mode.Sts_Maint) ] ,XIC(PCmd_Tare) [XIC(Cfg_PCmdClear) OTU(PCmd_Tare) ,NOP() ] XIC(Mode.Sts_Prog) ][XIO(Wrk_RunFlow) XIO(Wrk_BumpFlow) [XIO(Wrk_InpInfNaN) ,XIC(Inp_Sim) ] [OTL(Wrk_Tare) OTU(Wrk_BumpNoAdj) OTU(TareFault.Inp) ,OTU(OverTol.Inp) OTU(UnderTol.Inp) OTU(Sts_InTol) ,XIC(Inp_Sim) MOV(Cfg_SimStartWt,Wrk_PV) ,MOV(Wrk_PV,Wrk_TareWt) ] ,[XIC(Wrk_RunFlow) ,XIC(Wrk_BumpFlow) ,XIC(Wrk_InpInfNaN) XIO(Inp_Sim) ] OTL(TareFault.Inp) ];
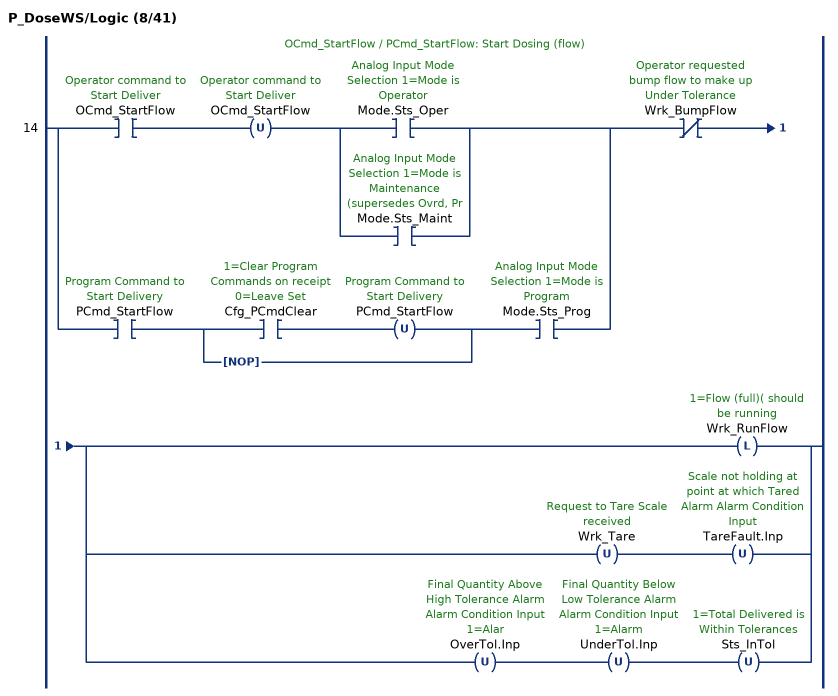
   // OCmd_StartFlow / PCmd_StartFlow: Start Dosing (flow)
   14: [XIC(OCmd_StartFlow) OTU(OCmd_StartFlow) [XIC(Mode.Sts_Oper) ,XIC(Mode.Sts_Maint) ] ,XIC(PCmd_StartFlow) [XIC(Cfg_PCmdClear) OTU(PCmd_StartFlow) ,NOP() ] XIC(Mode.Sts_Prog) ]XIO(Wrk_BumpFlow)[OTL(Wrk_RunFlow) ,OTU(Wrk_Tare) OTU(TareFault.Inp) ,OTU(OverTol.Inp) OTU(UnderTol.Inp) OTU(Sts_InTol) ];
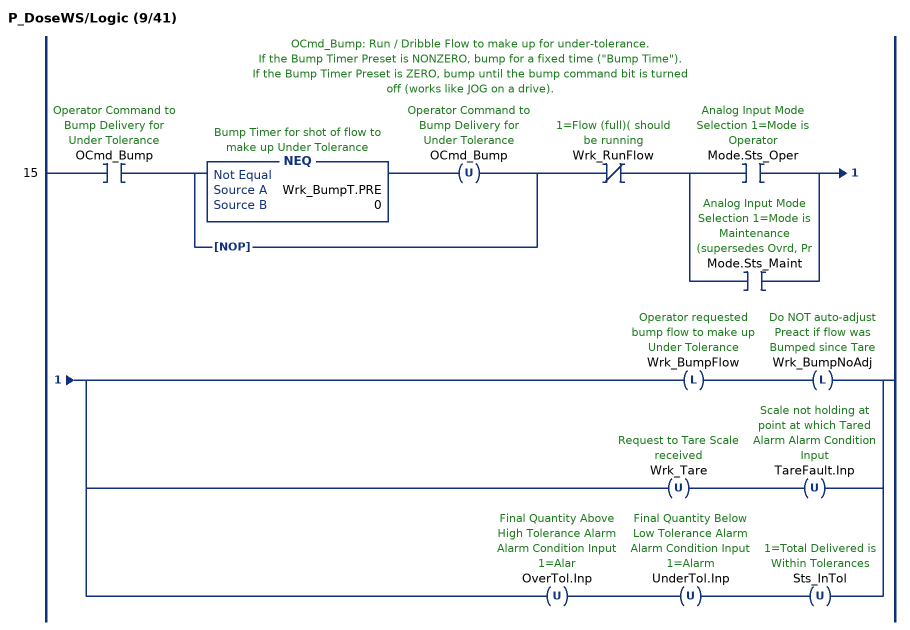
   // OCmd_Bump: Run / Dribble Flow to make up for under-tolerance.
   // If the Bump Timer Preset is NONZERO, bump for a fixed time ("Bump Time").
   // If the Bump Timer Preset is ZERO, bump until the bump command bit is turned
   // off (works like JOG on a drive).
   15: XIC(OCmd_Bump)[NEQ(Wrk_BumpT.PRE,0) OTU(OCmd_Bump) ,NOP() ]XIO(Wrk_RunFlow)[XIC(Mode.Sts_Oper) ,XIC(Mode.Sts_Maint) ][OTL(Wrk_BumpFlow) OTL(Wrk_BumpNoAdj) ,OTU(Wrk_Tare) OTU(TareFault.Inp) ,OTU(OverTol.Inp) OTU(UnderTol.Inp) OTU(Sts_InTol) ];
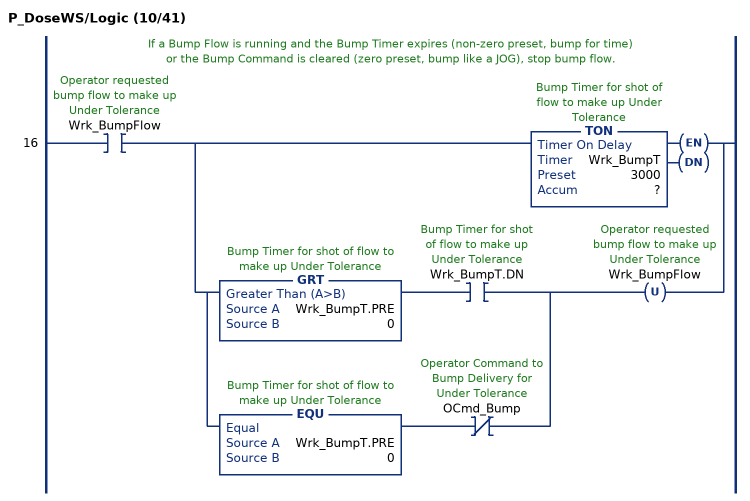
   // If a Bump Flow is running and the Bump Timer expires (non-zero preset, bump for time)
   // or the Bump Command is cleared (zero preset, bump like a JOG), stop bump flow.
   16: XIC(Wrk_BumpFlow)[TON(Wrk_BumpT,?,?) ,[GRT(Wrk_BumpT.PRE,0) XIC(Wrk_BumpT.DN) ,EQU(Wrk_BumpT.PRE,0) XIO(OCmd_Bump) ] OTU(Wrk_BumpFlow) ];
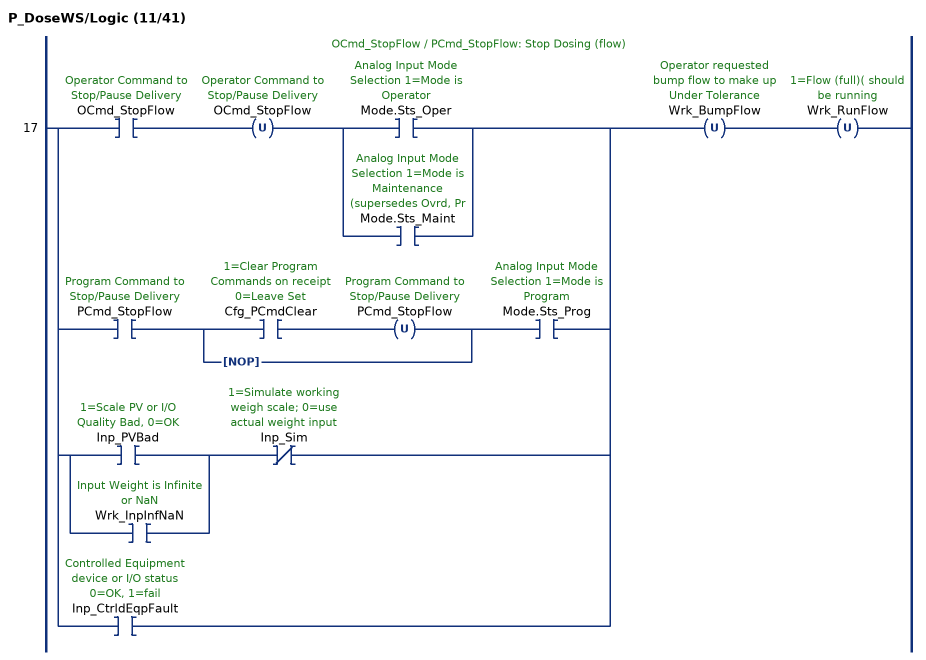
   // OCmd_StopFlow / PCmd_StopFlow: Stop Dosing (flow)
   17: [XIC(OCmd_StopFlow) OTU(OCmd_StopFlow) [XIC(Mode.Sts_Oper) ,XIC(Mode.Sts_Maint) ] ,XIC(PCmd_StopFlow) [XIC(Cfg_PCmdClear) OTU(PCmd_StopFlow) ,NOP() ] XIC(Mode.Sts_Prog) ,[XIC(Inp_PVBad) ,XIC(Wrk_InpInfNaN) ] XIO(Inp_Sim) ,XIC(Inp_CtrldEqpFault) ]OTU(Wrk_BumpFlow)OTU(Wrk_RunFlow);
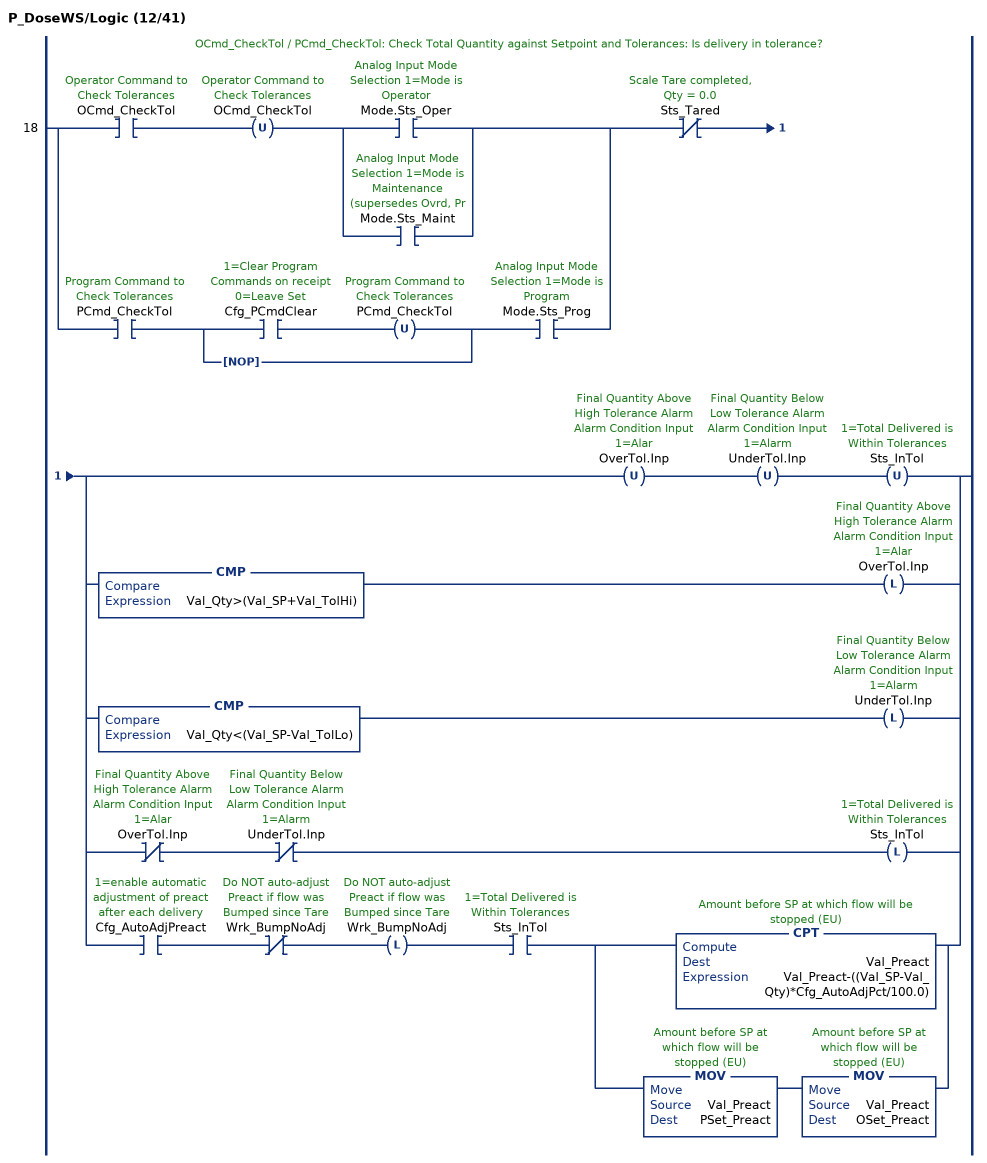
   // OCmd_CheckTol / PCmd_CheckTol: Check Total Quantity against Setpoint and Tolerances: Is delivery in tolerance?
   18: [XIC(OCmd_CheckTol) OTU(OCmd_CheckTol) [XIC(Mode.Sts_Oper) ,XIC(Mode.Sts_Maint) ] ,XIC(PCmd_CheckTol) [XIC(Cfg_PCmdClear) OTU(PCmd_CheckTol) ,NOP() ] XIC(Mode.Sts_Prog) ]XIO(Sts_Tared)[OTU(OverTol.Inp) OTU(UnderTol.Inp) OTU(Sts_InTol) ,CMP(Val_Qty>(Val_SP+Val_TolHi)) OTL(OverTol.Inp) ,CMP(Val_Qty<(Val_SP-Val_TolLo)) OTL(UnderTol.Inp) ,XIO(OverTol.Inp) XIO(UnderTol.Inp) OTL(Sts_InTol) ,XIC(Cfg_AutoAdjPreact) XIO(Wrk_BumpNoAdj) OTL(Wrk_BumpNoAdj) XIC(Sts_InTol) [CPT(Val_Preact,Val_Preact-((Val_SP-Val_Qty)*Cfg_AutoAdjPct/100.0)) ,MOV(Val_Preact,PSet_Preact) MOV(Val_Preact,OSet_Preact) ] ];
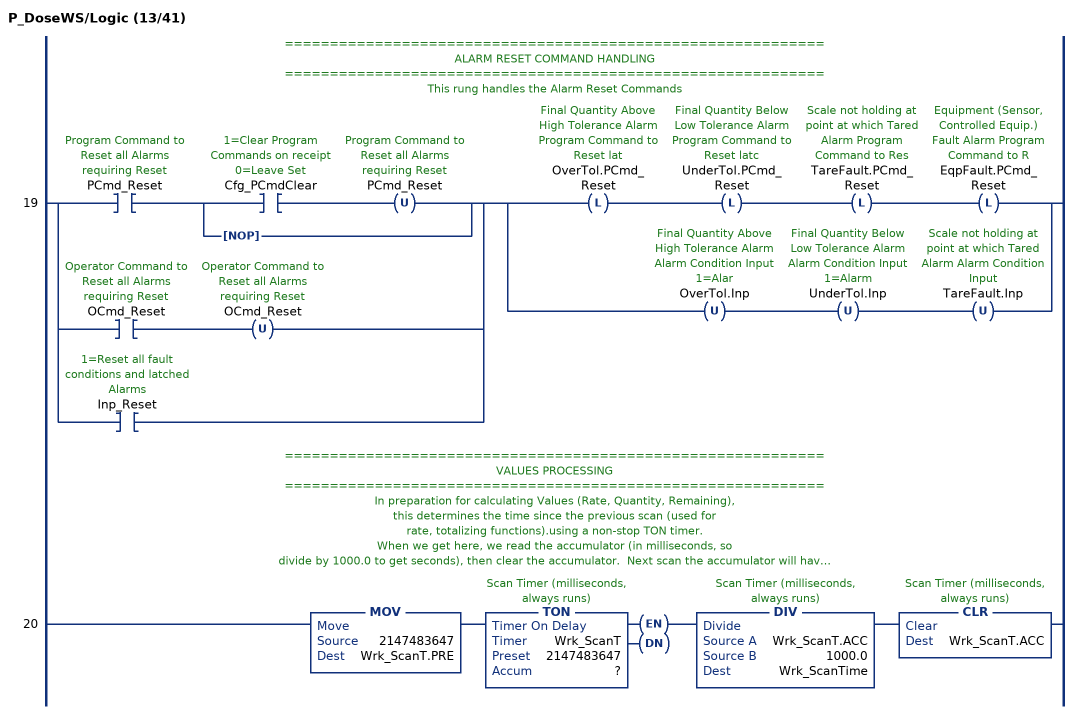
   // ============================================================
   // ALARM RESET COMMAND HANDLING
   // ============================================================
   // This rung handles the Alarm Reset Commands
   19: [XIC(PCmd_Reset) [XIC(Cfg_PCmdClear) OTU(PCmd_Reset) ,NOP() ] ,XIC(OCmd_Reset) OTU(OCmd_Reset) ,XIC(Inp_Reset) ][OTL(OverTol.PCmd_Reset) OTL(UnderTol.PCmd_Reset) OTL(TareFault.PCmd_Reset) OTL(EqpFault.PCmd_Reset) ,OTU(OverTol.Inp) OTU(UnderTol.Inp) OTU(TareFault.Inp) ];
   // ============================================================
   // VALUES PROCESSING
   // ============================================================
   // In preparation for calculating Values (Rate, Quantity, Remaining),
   // this determines the time since the previous scan (used for
   // rate, totalizing functions).using a non-stop TON timer.
   // When we get here, we read the accumulator (in milliseconds, so
   // divide by 1000.0 to get seconds), then clear the accumulator.  Next scan the accumulator will have
   // incremented up to the number of milliseconds since last scan.  (Works for scan times up to 2 million seconds.....)
   20: MOV(2147483647,Wrk_ScanT.PRE)TON(Wrk_ScanT,?,?)DIV(Wrk_ScanT.ACC,1000.0,Wrk_ScanTime)CLR(Wrk_ScanT.ACC);
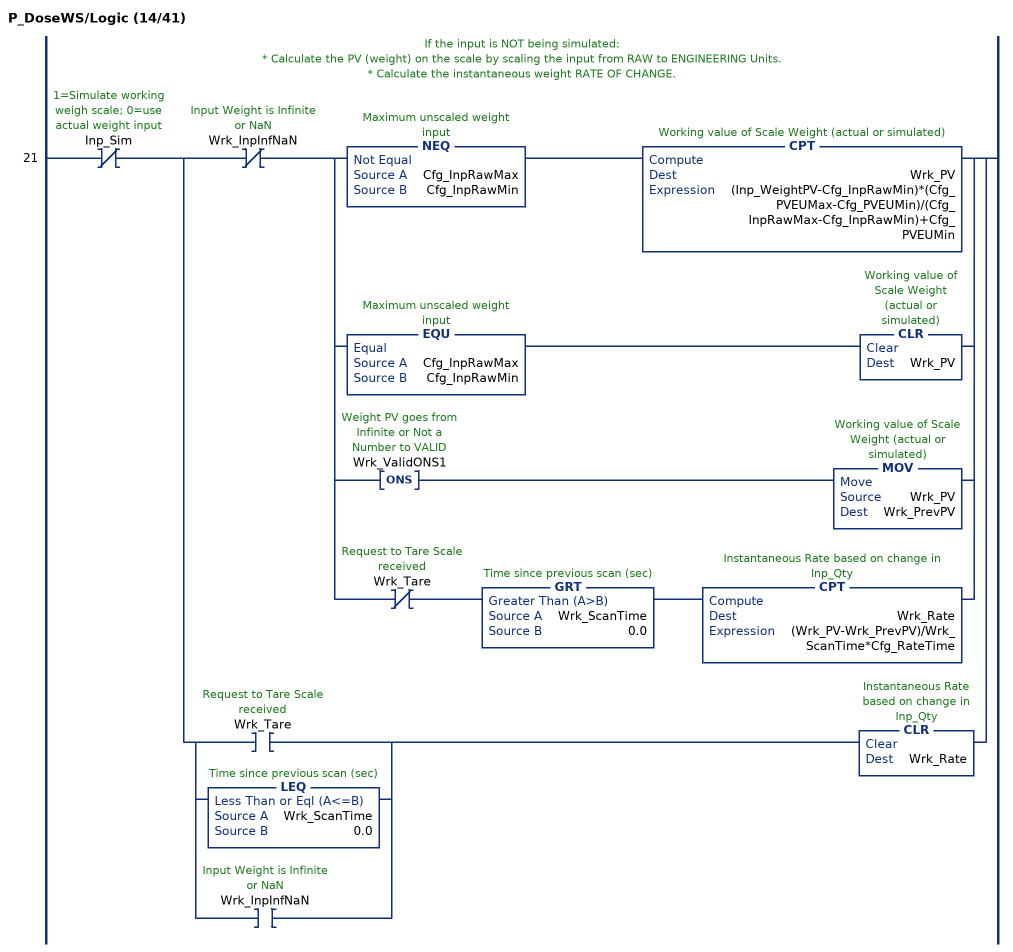
   // If the input is NOT being simulated:
   // * Calculate the PV (weight) on the scale by scaling the input from RAW to ENGINEERING Units.
   // * Calculate the instantaneous weight RATE OF CHANGE.
   21: XIO(Inp_Sim)[XIO(Wrk_InpInfNaN) [NEQ(Cfg_InpRawMax,Cfg_InpRawMin) CPT(Wrk_PV,(Inp_WeightPV-Cfg_InpRawMin)*(Cfg_PVEUMax-Cfg_PVEUMin)/(Cfg_InpRawMax-Cfg_InpRawMin)+Cfg_PVEUMin) ,EQU(Cfg_InpRawMax,Cfg_InpRawMin) CLR(Wrk_PV) ,ONS(Wrk_ValidONS1) MOV(Wrk_PV,Wrk_PrevPV) ,XIO(Wrk_Tare) GRT(Wrk_ScanTime,0.0) CPT(Wrk_Rate,(Wrk_PV-Wrk_PrevPV)/Wrk_ScanTime*Cfg_RateTime) ] ,[XIC(Wrk_Tare) ,LEQ(Wrk_ScanTime,0.0) ,XIC(Wrk_InpInfNaN) ] CLR(Wrk_Rate) ];
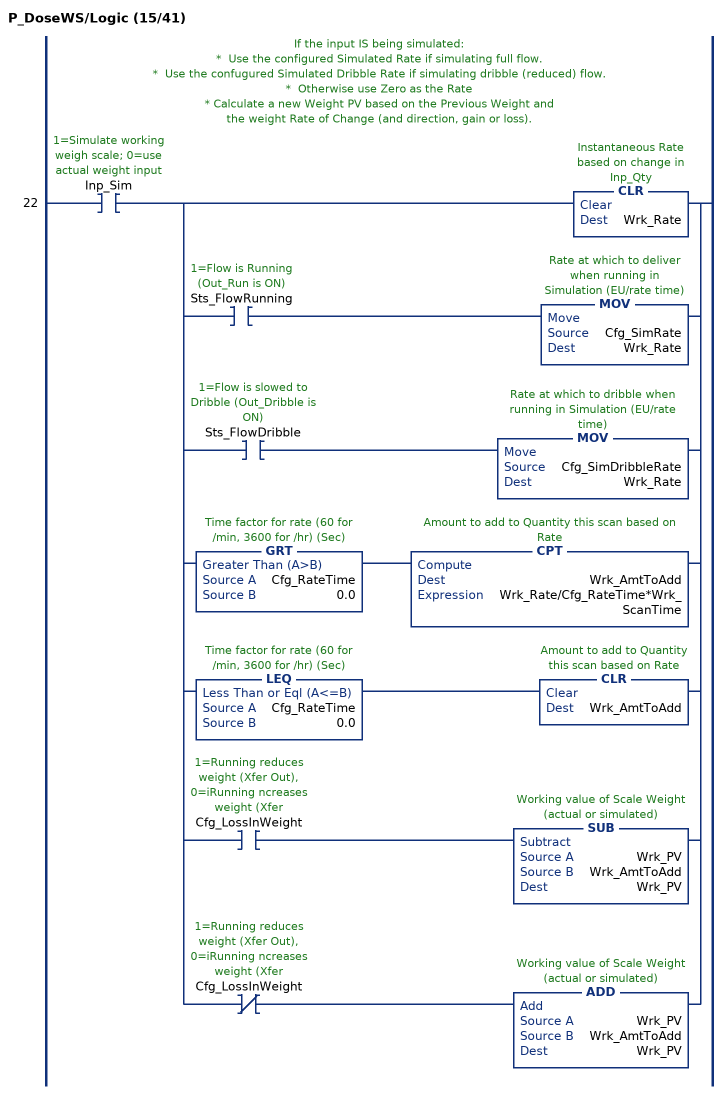
   // If the input IS being simulated:
   // *  Use the configured Simulated Rate if simulating full flow.
   // *  Use the confugured Simulated Dribble Rate if simulating dribble (reduced) flow.
   // *  Otherwise use Zero as the Rate
   // * Calculate a new Weight PV based on the Previous Weight and
   // the weight Rate of Change (and direction, gain or loss).
   22: XIC(Inp_Sim)[CLR(Wrk_Rate) ,XIC(Sts_FlowRunning) MOV(Cfg_SimRate,Wrk_Rate) ,XIC(Sts_FlowDribble) MOV(Cfg_SimDribbleRate,Wrk_Rate) ,GRT(Cfg_RateTime,0.0) CPT(Wrk_AmtToAdd,Wrk_Rate/Cfg_RateTime*Wrk_ScanTime) ,LEQ(Cfg_RateTime,0.0) CLR(Wrk_AmtToAdd) ,XIC(Cfg_LossInWeight) SUB(Wrk_PV,Wrk_AmtToAdd,Wrk_PV) ,XIO(Cfg_LossInWeight) ADD(Wrk_PV,Wrk_AmtToAdd,Wrk_PV) ];
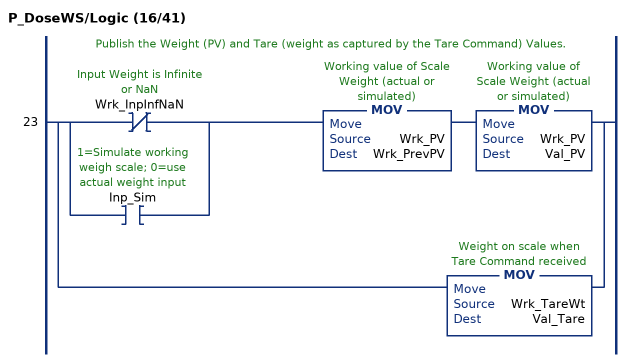
   // Publish the Weight (PV) and Tare (weight as captured by the Tare Command) Values.
   23: [[XIO(Wrk_InpInfNaN) ,XIC(Inp_Sim) ] MOV(Wrk_PV,Wrk_PrevPV) MOV(Wrk_PV,Val_PV) ,MOV(Wrk_TareWt,Val_Tare) ];
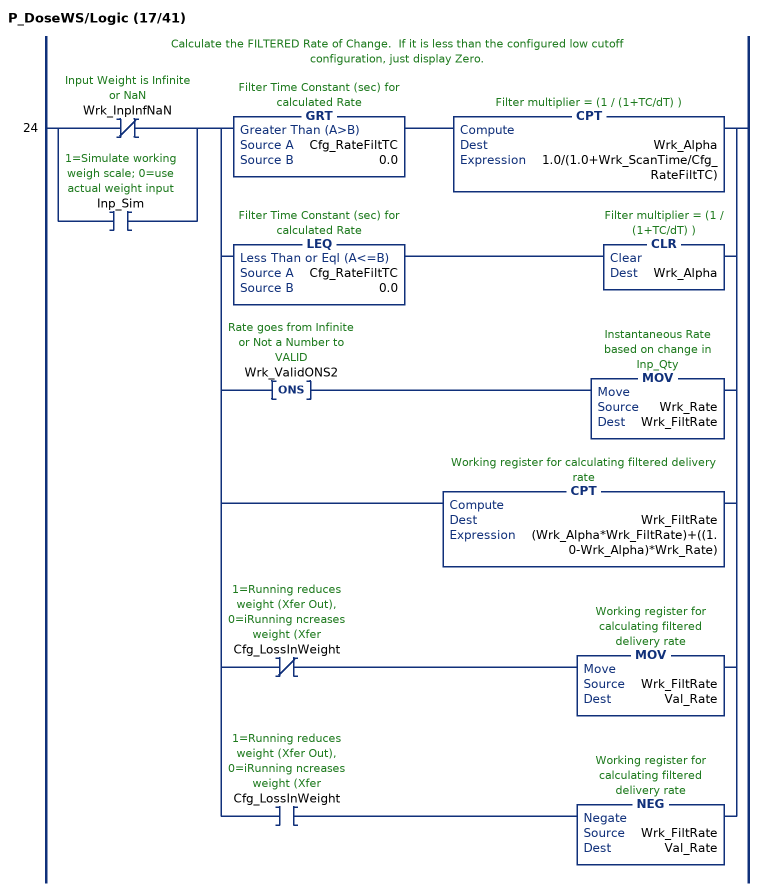
   // Calculate the FILTERED Rate of Change.  If it is less than the configured low cutoff
   // configuration, just display Zero.
   24: [XIO(Wrk_InpInfNaN) ,XIC(Inp_Sim) ][GRT(Cfg_RateFiltTC,0.0) CPT(Wrk_Alpha,1.0/(1.0+Wrk_ScanTime/Cfg_RateFiltTC)) ,LEQ(Cfg_RateFiltTC,0.0) CLR(Wrk_Alpha) ,ONS(Wrk_ValidONS2) MOV(Wrk_Rate,Wrk_FiltRate) ,CPT(Wrk_FiltRate,(Wrk_Alpha*Wrk_FiltRate)+((1.0-Wrk_Alpha)*Wrk_Rate)) ,XIO(Cfg_LossInWeight) MOV(Wrk_FiltRate,Val_Rate) ,XIC(Cfg_LossInWeight) NEG(Wrk_FiltRate,Val_Rate) ];
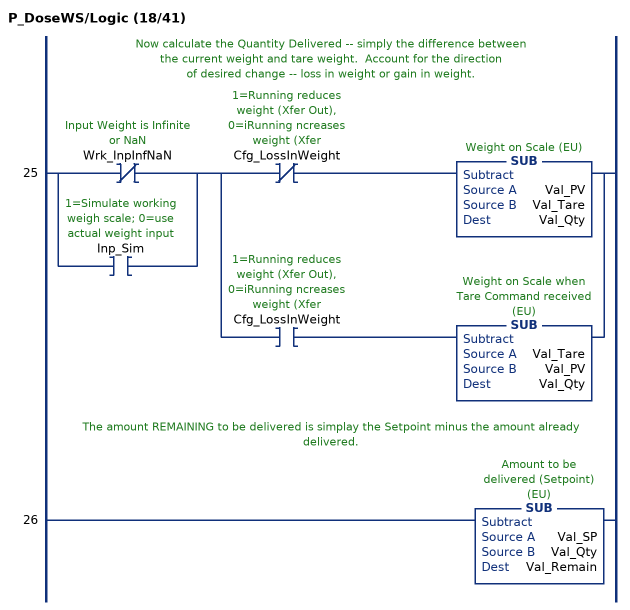
   // Now calculate the Quantity Delivered -- simply the difference between
   // the current weight and tare weight.  Account for the direction
   // of desired change -- loss in weight or gain in weight.
   25: [XIO(Wrk_InpInfNaN) ,XIC(Inp_Sim) ][XIO(Cfg_LossInWeight) SUB(Val_PV,Val_Tare,Val_Qty) ,XIC(Cfg_LossInWeight) SUB(Val_Tare,Val_PV,Val_Qty) ];
   // The amount REMAINING to be delivered is simplay the Setpoint minus the amount already delivered.
   26: SUB(Val_SP,Val_Qty,Val_Remain);
